{attribute 'qualified_only'}
{attribute 'strict'}
TYPE Homing :
(
	IDLE,
	
	START,
	RETRY,
	
	STOP,
	SET,
	DONE,
	
	size
);
END_TYPE
(*
general homing sequence:
	on drive.homingSequence() call, home towards home sensor
	if home reached, set position and finish homing as usual
	if outer limit reached, traverse towards inner limit
		when inner limit reached, retry homing
*)

(* stored: Version 1.1.0.1, ProductVersion 3.1.4024.11
   DUT Homing: Id {bf7a16b6-9b16-4fc3-90d5-848d709e6d7e} *)
